PROGRAM MAIN
VAR	
END_VAR

//Hannes Viljamaa
motor();
light();
control();
blinker();
//Hardware();

END_PROGRAM

(* stored: Version 1.1.0.1, ProductVersion 3.1.4024.11
   POU MAIN: Id {0d037d36-53d9-4a5a-a763-1819dd5d0f00}, SpecialFunc None *)
